FUNCTION_BLOCK TcCamTable IMPLEMENTS itfCamTable
VAR_INPUT
END_VAR
VAR_OUTPUT
END_VAR
VAR
END_VAR

{warning 'add method implementation '}
METHOD Select 		: itfCommand
VAR_INPUT	
	Periodic		: BOOL;
	MasterAbsolute	: BOOL;
	SlaveAbsolute	: BOOL;
	CamTable		: MC_CAM_REF;
END_VAR
VAR
	
END_VAR
END_METHOD

END_FUNCTION_BLOCK

(* stored: Version 1.1.0.1, ProductVersion 3.1.4024.12
   POU TcCamTable: Id {c488141e-f0f7-4f2f-8107-b3f60bfb46cb}, SpecialFunc None
   Method Select: Id {7b02621f-18e7-43c8-9b84-9b4a4588b20c} *)
